PROGRAM MAIN

VAR

END_VAR

P_Inputs();
P_MachineControl();
P_AxisControl();
P_Outputs();
P_StablePlatform();

END_PROGRAM

(* stored: Version 1.1.0.1, ProductVersion 3.1.4024.12
   POU MAIN: Id {540b8970-e57b-4c7b-a65e-22bf2965a9b1}, SpecialFunc None *)
